(* Logix 5000 project; controller Convert Emulate 5570 rev 36.11; software revision 36.00 *)

TASK MainTask (continuous, watchdog 500 ms) : MainProgram

MODULES
   Local : Emulate 5570 (ICP 2, rev 36.11)
       : 1756-IB16 (ICP 3, rev 3.1, Input RPI 20 ms)
       : 1756-IB16 (ICP 5, rev 3.1, Input RPI 20 ms)
       : vendor 1 type 7 code 16 (ICP 4, rev 3.1, Output RPI 20 ms)
END_MODULES

VAR_GLOBAL   (* controller tags *)
   CONVERT_PB : ALIAS FOR Local:3:I.Data.14;   // Convert Temperature N.O. Pushbutton
   ERROR_DUP_VAL : ALIAS FOR Local:4:O.Data.0;   // Error Duplicate Value Indicator
   ERROR_OVER_VAL : ALIAS FOR Local:4:O.Data.1;   // Data Error, Over Value
   H_INDC : ALIAS FOR Local:4:O.Data.5;   // High Indicator
   HH_INDC : ALIAS FOR Local:4:O.Data.6;   // High High Indicator
   L_INDC : ALIAS FOR Local:4:O.Data.3;   // Low Indicator
   LL_INDC : ALIAS FOR Local:4:O.Data.2;   // Low Low Indicator
   M_INDC : ALIAS FOR Local:4:O.Data.4;   // Mid Indicator
   RESET_PB : ALIAS FOR Local:3:I.Data.15;   // Data Error Reset, N.O. Pushbutton
   TWS_INPUT : ALIAS FOR Local:5:I.Data;   // Thumbwheel Switch, Celsius Value
END_VAR

PROGRAM MainProgram   (* main routine MainRoutine *)
VAR
   C_TEMP : DINT := 64;   // Celsius Temperature
   C_TEMP_CONVERT : DINT := 64;   // Celsius Temperature Parameter
   C_TEMP_STORAGE : DINT := 64;   // Storage of Celsius Temperature
   DIV_RESULT : DINT := 115;   // Divide Result
   F_TEMP : DINT := 147;   // Fahrenheit Value
   F_TEMP_CONVERT : DINT := 147;   // Fahrenheit Temperature Parameter
   HMI_CONVERT_PB : BOOL;   // HMI Convert Button
   HMI_ENABLE_DISABLE : BOOL := 1;   // HMI Enable/Disable Button
   HMI_RESET_PB : BOOL;   // HMI Reset Button
   INTERNAL_CONVERT : BOOL;   // Internal Control, Enable Convert
   MUL_RESULT : DINT := 576;   // Multiply Result
   ONE_SHOT_CONTROL : BOOL;   // One Shot
END_VAR

ROUTINE ConvertRoutine   (* ladder *)
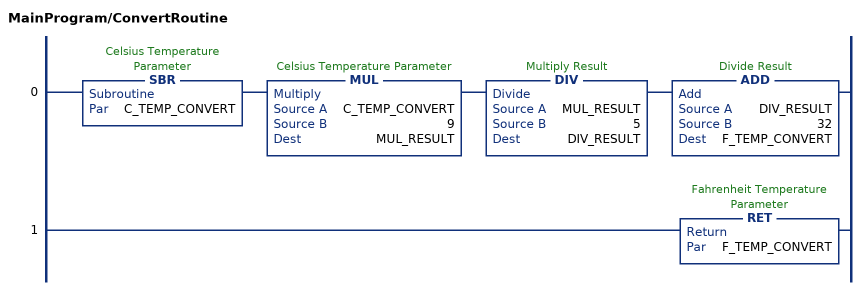
   0: SBR(C_TEMP_CONVERT)MUL(C_TEMP_CONVERT,9,MUL_RESULT)DIV(MUL_RESULT,5,DIV_RESULT)ADD(DIV_RESULT,32,F_TEMP_CONVERT);
   1: RET(F_TEMP_CONVERT);
END_ROUTINE

ROUTINE IndicatorsRoutine   (* ladder *)
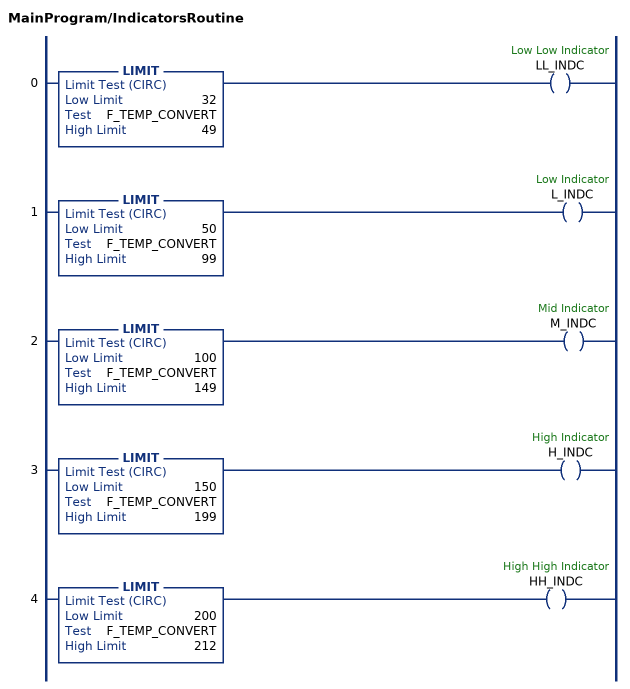
   0: LIMIT(32,F_TEMP_CONVERT,49)OTE(LL_INDC);
   1: LIMIT(50,F_TEMP_CONVERT,99)OTE(L_INDC);
   2: LIMIT(100,F_TEMP_CONVERT,149)OTE(M_INDC);
   3: LIMIT(150,F_TEMP_CONVERT,199)OTE(H_INDC);
   4: LIMIT(200,F_TEMP_CONVERT,212)OTE(HH_INDC);
END_ROUTINE

ROUTINE InputControlRoutine   (* ladder *)
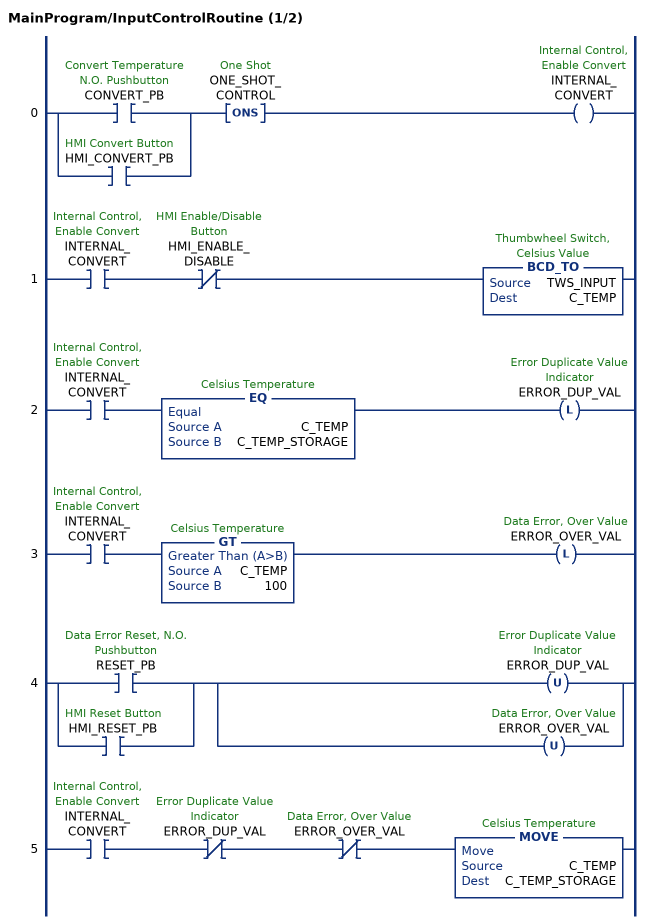
   0: [XIC(CONVERT_PB) ,XIC(HMI_CONVERT_PB) ]ONS(ONE_SHOT_CONTROL)OTE(INTERNAL_CONVERT);
   1: XIC(INTERNAL_CONVERT)XIO(HMI_ENABLE_DISABLE)BCD_TO(TWS_INPUT,C_TEMP);
   2: XIC(INTERNAL_CONVERT)EQ(C_TEMP,C_TEMP_STORAGE)OTL(ERROR_DUP_VAL);
   3: XIC(INTERNAL_CONVERT)GT(C_TEMP,100)OTL(ERROR_OVER_VAL);
   4: [XIC(RESET_PB) ,XIC(HMI_RESET_PB) ][OTU(ERROR_DUP_VAL) ,OTU(ERROR_OVER_VAL) ];
   5: XIC(INTERNAL_CONVERT)XIO(ERROR_DUP_VAL)XIO(ERROR_OVER_VAL)MOVE(C_TEMP,C_TEMP_STORAGE);
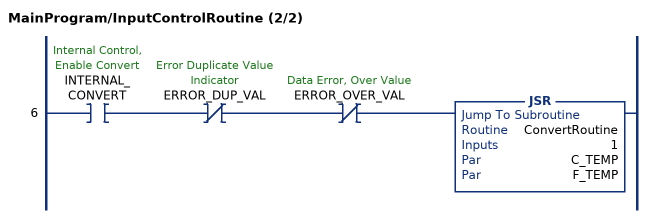
   6: XIC(INTERNAL_CONVERT)XIO(ERROR_DUP_VAL)XIO(ERROR_OVER_VAL)JSR(ConvertRoutine,1,C_TEMP,F_TEMP);
END_ROUTINE

ROUTINE MainRoutine   (* ladder *)
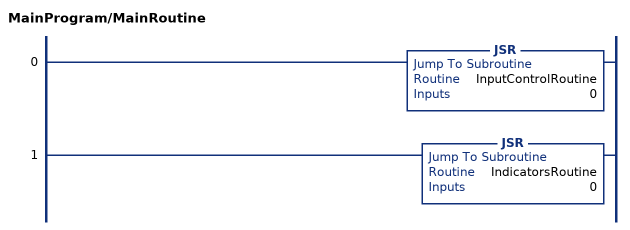
   0: JSR(InputControlRoutine,0);
   1: JSR(IndicatorsRoutine,0);
END_ROUTINE
END_PROGRAM
